{attribute 'qualified_only'}
{attribute 'strict'}
{attribute 'to_string'}
TYPE E_MaterialServiceErrorCode :
(
	None := 0,
	InvalidCommand := 900,
	TargetEndpointIdRequired := 901,
	TargetEndpointNotFound := 902,
	DuplicateTargetEndpointId := 903
) UDINT;
END_TYPE

(* stored: Version 1.1.0.1, ProductVersion 3.1.4026.18
   DUT E_MaterialServiceErrorCode: Id {6c8fb4a8-f244-4036-9d41-088e65757441} *)
